FUNCTION_BLOCK OpticSensor (* Template for an empty basic function block *)
  (* Standard: 61499-2 *)
  (* Version 1.0, 2019-03-19, Duc Do Tran, OFFIS e.V. *)
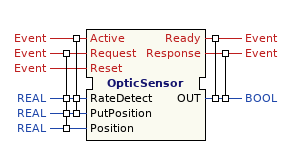
  EVENT_INPUT
    Active WITH RateDetect, PutPosition;
    Request WITH RateDetect, PutPosition, Position;
    Reset;
  END_EVENT
  EVENT_OUTPUT
    Ready WITH OUT;
    Response WITH OUT;
  END_EVENT
  VAR_INPUT
    RateDetect : REAL := 0.001;
    PutPosition : REAL := 180;
    Position : REAL;
  END_VAR
  VAR_OUTPUT
    OUT : BOOL := FALSE;
  END_VAR
  VAR
    trigger : BOOL; (* Internal Variable *)
    change : BOOL; (* Internal Variable *)
  END_VAR
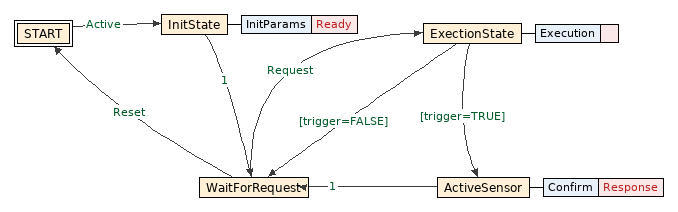
  EC_STATES
    START; (* Initial State *)
    ActiveSensor : Confirm -> Response;
    ExectionState : Execution;
    InitState : InitParams -> Ready;
    WaitForRequest;
  END_STATES
  EC_TRANSITIONS
    ExectionState TO WaitForRequest := [trigger=FALSE];
    ExectionState TO ActiveSensor := [trigger=TRUE];
    START TO InitState := Active;
    WaitForRequest TO ExectionState := Request;
    ActiveSensor TO WaitForRequest := 1;
    WaitForRequest TO START := Reset;
    InitState TO WaitForRequest := 1;
  END_TRANSITIONS
  ALGORITHM Confirm IN ST: (* new algorithm *)
OUT := TRUE;
trigger := FALSE;
  END_ALGORITHM
  ALGORITHM Execution IN ST: (* new algorithm *)
IF ((Position >= PutPosition*(1-RateDetect)) AND (Position <= PutPosition*(1+RateDetect))) THEN
	IF (change = FALSE) THEN
		change := TRUE;
		trigger := TRUE;
	END_IF;
ELSE
	IF (change = TRUE) THEN
		change := FALSE;
		OUT := FALSE;
	END_IF;
	trigger := FALSE;
END_IF;
  END_ALGORITHM
  ALGORITHM InitParams IN ST: (* new algorithm *)
OUT := FALSE;
trigger := FALSE;
change := FALSE;
  END_ALGORITHM
END_FUNCTION_BLOCK
